// TIA Portal V17 export
// export: Created 2025-06-25T13:13:23.1608213Z, ExportSetting WithDefaults, DisplayName Totally Integrated Automation Portal, DisplayVersion V17 Update 8, DisplayName TIA Portal Openness, DisplayVersion V17 Update 8, DisplayName TIA Portal Version Control Interface, DisplayVersion V17, DisplayName STEP 7 Professional, DisplayVersion V17 Update 8, DisplayName STEP 7 Safety, DisplayVersion V17 Update 6, DisplayName WinCC Advanced, DisplayVersion V17 Update 8
FUNCTION_BLOCK "fbHighAlarm"   // FB31, FBD
TITLE = Lightweight version of fbAnalogAlarm with only one limit
{ S7_Optimized_Access := 'TRUE' }
VERSION : 0.1
// stored: AutoNumber true, IsIECCheckEnabled false, IsRetainMemResEnabled false, MemoryReserve 0, SetENOAutomatically false, UDAEnableTagReadback false
   VAR_INPUT
      sValue : "stCalcValue";
      bAckAll : Bool;
      bEnable : Bool;
   END_VAR
   VAR_IN_OUT
      sTag : "stLimitAlarm";
   END_VAR
   VAR
      Alarm : "fbLimitAlarm";
   END_VAR
   VAR CONSTANT
      Low : Bool;
      High : Bool := true;
   END_VAR
BEGIN

REGION Network 1
   // Note that alarm is disabled if CalcValue .bError is set
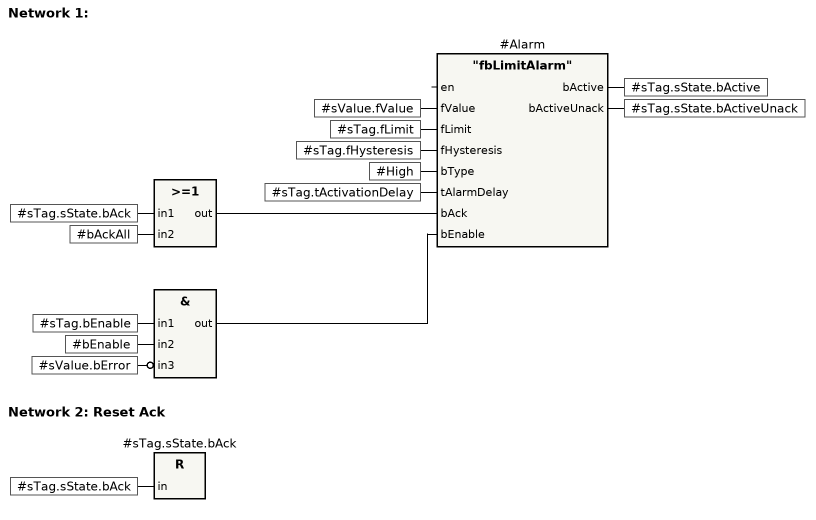
   #Alarm(fValue := #sValue.fValue,   // "fbLimitAlarm"
          fLimit := #sTag.fLimit,
          fHysteresis := #sTag.fHysteresis,
          bType := #High,
          tAlarmDelay := #sTag.tActivationDelay,
          bAck := #sTag.sState.bAck OR #bAckAll,
          bEnable := #sTag.bEnable AND #bEnable AND NOT #sValue.bError,
          bActive => #sTag.sState.bActive,
          bActiveUnack => #sTag.sState.bActiveUnack);
END_REGION

REGION Network 2: Reset Ack
   IF #sTag.sState.bAck THEN #sTag.sState.bAck := FALSE; END_IF;
END_REGION
END_FUNCTION_BLOCK
